FUNCTION TryConvert_DWORD_TO_TOD : BOOL
VAR_INPUT
	in : DWORD;
	out : REFERENCE TO TOD;
END_VAR

IF in > DatatypeLimits.MAX_VALUE_OF_DWORD_WHICH_CAN_BE_HELD_IN_A_TOD THEN
	RETURN;
END_IF

out := DWORD_TO_TOD(in);
TryConvert_DWORD_TO_TOD := TRUE;

END_FUNCTION

(* stored: Version 1.1.0.1, ProductVersion 3.1.4024.12
   POU TryConvert_DWORD_TO_TOD: Id {a0c1d43f-3422-484d-9996-357d6e83a34e}, SpecialFunc None *)
